FUNCTION_BLOCK TableSerializer
VAR
	_StringBuilder : REFERENCE TO StringBuilderExtBuffer;
	
	rowDefinition : __SYSTEM.AnyType;
	_RowCount : DINT;
	_ColumnDefinitionBuffer : ARRAY[0..MaxColumnCount - 1] OF __SYSTEM.AnyType;
	_ColumnNameBuffer : ARRAY[0..MaxColumnCount - 1] OF T_MaxString;
	definedColumns : INT;
	
	_Separator : STRING := ','; // Default separator ';' is compatible with european decimal separator '.'.
	_NewLine : STRING := '$N'; // Default is Windows newline.
	_DecimalSeparator : STRING := '.';
END_VAR
VAR CONSTANT
	MaxColumnCount : INT := TableSerializationParameters.SerializerMaxColumns;
	DefaultDecimalSeparator : STRING := '.';
END_VAR

METHOD PRIVATE AddColumnHeader
VAR
	column : INT;
END_VAR
FOR column := 0 TO definedColumns - 1 DO
	IF (column > 0) THEN
		_StringBuilder.Append(_Separator);
	END_IF
	
	_StringBuilder.Append(_ColumnNameBuffer[column]);
END_FOR
END_METHOD

METHOD PRIVATE AddLine
VAR_INPUT
	rowIndex : DINT;
END_VAR
VAR
	column : INT;
	currentData : __SYSTEM.AnyType;
	converted : T_MaxString;
END_VAR
FOR column := 0 TO definedColumns - 1 DO
	IF (column > 0) THEN
		_StringBuilder.Append(_Separator);
	END_IF
	
	currentData := _ColumnDefinitionBuffer[column];
	currentData.pValue := rowDefinition.pValue + TO_DWORD(rowDefinition.diSize * rowIndex) + (currentData.pValue - rowDefinition.pValue);
	
	IF (TO_INT(currentData.TypeClass) = IBaseLibrary.TypeClass.TYPE_STRING) THEN
		_StringBuilder.AppendByPointer(currentData.pValue);
	ELSE
		converted := AnyTypeToString(currentData);
		
		CASE TO_INT(currentData.TypeClass) OF
			TYPE_REAL, TYPE_LREAL:
				ReplaceString(converted, DefaultDecimalSeparator, _DecimalSeparator);
		END_CASE
		
		_StringBuilder.Append(converted);
	END_IF
END_FOR
END_METHOD

METHOD PRIVATE AddNewLine
_StringBuilder.Append(_NewLine);
END_METHOD

METHOD PRIVATE AddRows
VAR
	row : DINT;
END_VAR
FOR row := 0 TO _RowCount - 1 DO
	IF (row > 0) THEN
		AddNewLine();
	END_IF
	AddLine(row);
END_FOR
END_METHOD

{attribute 'monitoring' := 'call'}
PROPERTY DecimalSeparator : STRING
GET
DecimalSeparator := _DecimalSeparator;
END_GET
SET
_DecimalSeparator := DecimalSeparator;
END_SET
END_PROPERTY

METHOD DefineNextColumn : REFERENCE TO TableSerializer
VAR_INPUT
	columnInFirstRow : ANY; 
END_VAR
IF (definedColumns < MaxColumnCount) THEN
	_ColumnDefinitionBuffer[definedColumns] := columnInFirstRow;
	definedColumns := definedColumns + 1;
END_IF

DefineNextColumn REF= THIS^;
END_METHOD

METHOD DefineNextColumnWithName : REFERENCE TO TableSerializer
VAR_INPUT
	columnInFirstRow : ANY;
	name : T_MaxString;
END_VAR
IF (definedColumns < MaxColumnCount) THEN
	_ColumnDefinitionBuffer[definedColumns] := columnInFirstRow;
	_ColumnNameBuffer[definedColumns] := name;
	definedColumns := definedColumns + 1;
END_IF

DefineNextColumnWithName REF= THIS^;
END_METHOD

METHOD DefineRow : REFERENCE TO TableSerializer
VAR_INPUT
	firstRow : ANY;
END_VAR
rowDefinition := firstRow;

DefineRow REF= THIS^;
END_METHOD

{attribute 'monitoring' := 'call'}
PROPERTY NewLine : STRING
GET
NewLine := _NewLine;
END_GET
SET
_NewLine := NewLine;
END_SET
END_PROPERTY

{attribute 'monitoring' := 'call'}
PROPERTY RowCount : DINT
GET
RowCount := _RowCount;
END_GET
SET
_RowCount := RowCount;
END_SET
END_PROPERTY

{attribute 'monitoring' := 'call'}
PROPERTY Separator : STRING
GET
Separator := _Separator;
END_GET
SET
_Separator := Separator;
END_SET
END_PROPERTY

METHOD Serialize
VAR_INPUT
	includeHeader : BOOL;
	clearBuffer : BOOL;
END_VAR
IF (clearBuffer) THEN
	_StringBuilder.Clear();
END_IF
IF (includeHeader) THEN
	AddColumnHeader();
	AddNewLine();
END_IF
AddRows();
END_METHOD

{attribute 'monitoring' := 'call'}
PROPERTY SerializedLength : DINT
GET
SerializedLength := _StringBuilder.Length;
END_GET
END_PROPERTY

{attribute 'monitoring' := 'call'}
PROPERTY SerializedString : POINTER TO STRING
GET
SerializedString := stringBuilder.BufferRef.pValue;
END_GET
END_PROPERTY

{attribute 'monitoring' := 'call'}
PROPERTY StringBuilder : REFERENCE TO StringBuilderExtBuffer
GET
StringBuilder REF= _StringBuilder;
END_GET
SET
_StringBuilder REF= StringBuilder;
END_SET
END_PROPERTY

END_FUNCTION_BLOCK

(* stored: Version 1.1.0.1
   POU TableSerializer: Id {d72633b8-404b-0f0c-3a80-0e4530f50430}, SpecialFunc None
   Method AddColumnHeader: Id {a96e7383-fed6-092f-1ef5-a1a0885e5cef}
   Method AddLine: Id {d9b58cd7-c635-083b-245e-5fb2dcc20db1}
   Method AddNewLine: Id {8ec85cae-9933-0793-348f-1132550fb9cc}
   Method AddRows: Id {38ae6eb7-6156-043d-0e52-11eeb0fae8ae}
   Property DecimalSeparator: Id {e0d5ba62-8fd6-40b3-9562-489e5ddaa896}
   Get Get: Id {8ea79d6a-2342-0545-2cc0-e4e91166ef27}
   Set Set: Id {80a9824f-9b84-0d64-3268-84dbb3923f5f}
   Method DefineNextColumn: Id {0973f48c-2795-0d69-1d24-997b7f4e2c7c}
   Method DefineNextColumnWithName: Id {2f43709f-d72d-479f-9470-44678b62a170}
   Method DefineRow: Id {ce8b20c5-e365-0d17-3c1b-aff8c931bd36}
   Property NewLine: Id {f3191bed-a76c-497f-9870-657f833967bb}
   Get Get: Id {ad21bc57-fed1-00cc-1f46-a3e827e39338}
   Set Set: Id {a329f98b-5509-0429-0983-71e2f9448074}
   Property RowCount: Id {3e6b6630-8c3b-04e2-1eba-68e455e01a12}
   Get Get: Id {b06bd905-8290-00fb-041b-5e64a8ce6802}
   Set Set: Id {620d98a1-8b4c-0a2a-1f03-9902bb377224}
   Property Separator: Id {8cc3ea40-abc9-03a0-0a4f-104f98552394}
   Get Get: Id {9324c3eb-b7b7-0ad9-16d5-2297110192ec}
   Set Set: Id {1ecb02ec-8f8c-0059-152f-75162282ff7d}
   Method Serialize: Id {3fe63765-60b0-0c99-3c86-f4191a72f13d}
   Property SerializedLength: Id {0c3ff8d0-5998-0d93-0787-87bbcb89aa15}
   Get Get: Id {1dbe863d-9a29-05a4-02ae-9be499a26d02}
   Property SerializedString: Id {8c948389-713e-0c66-1d60-1dadcc7a4b0c}
   Get Get: Id {e81efac8-b87a-0f5c-0835-40a8ed332183}
   Property StringBuilder: Id {39124655-37bb-4d64-951c-e421cd348791}
   Get Get: Id {87dabea9-c665-4b57-989c-177415199184}
   Set Set: Id {b7a571a6-05c2-44cf-a574-e55d3061e06c} *)
